// TIA Portal V16 export
// export: Created 2021-04-12T08:07:26.5150584Z, ExportSetting WithDefaults, DisplayName Totally Integrated Automation Portal, DisplayVersion V16, DisplayName TIA Portal Version Control Interface, DisplayVersion V16, DisplayName TIA Portal Openness, DisplayVersion V16, DisplayName STEP 7 Professional, DisplayVersion V16, DisplayName STEP 7 Safety, DisplayVersion V16, DisplayName WinCC Unified SCADA Engineering System, DisplayVersion V16
DATA_BLOCK "AutoMode_DB"   // DB5
VERSION : 0.1
// stored: AutoNumber true, DBAccessibleFromOPCUA true, InstanceOfName AutoMode, InstanceOfType FB
"AutoMode"
   // VAR_IN_OUT
   //    enableAutoMode : Bool;
   //    isFinishPreWork : Bool;
   //    isStartAutoMode : Bool;
   // END_VAR
   // VAR
   //    TaskSetWeight : Real;
   //    SetWeightBunker : Array[0..12] of Real;
   //    currentWeightBunker : Array[0..12] of Real;
   //    readyToSort : Array[0..12] of Bool;
   //    readyToDrop : Array[0..12] of Bool;
   //    readyToDropYP : Array[0..2] of Bool;
   //    isWorkWithBunker : Array[0..12] of Bool;
   //    preWorkAutoMode : Struct
   //       isFinishPreWork : Bool;
   //       alarmStop : Bool;
   //    END_STRUCT;
   //    preWork_AM_FB : "preWork_AM";
   //    workPackingMachine_AM_FB : "workPackingMachine_AM";
   //    workInConveyer_AM_FB : "workInConveyer_AM";
   //    controlFllipper_AM_FB : "controlValve";
   //    workVibroLot_AM_FB : Array[0..12] of "workVibroLot_AM";
   //    workVibroTable_AM_FB : "workVibroTable_AM";
   //    weightModule_AM_FB : "weightModule_AM";
   //    Sorting_AM_FB : "Sorting_AM";
   //    setWeightBunker_FB : "setWeightBunker_AM";
   //    blockSorting : Bool;
   //    openFlipper : Bool;
   //    hmiYpDropWeight : Array[0..2] of Real;
   //    hmiYpDropError : Array[0..2] of Real;
   //    Sorting_AM_withBuffer_FB { S7_SetPoint := 'True'} : "Sorting_AM_withBuffer";
   // END_VAR
BEGIN
END_DATA_BLOCK
